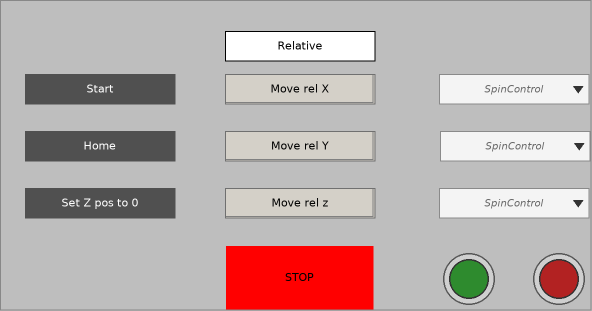
VISUALIZATION goPositionRel  // 592x311
    Button (225,74 150x30), "Move rel X"
        tap POSITION.DoRel_X
    Button (225,131 150x30), "Move rel Y"
        tap POSITION.DoRel_Y
    Button (225,188 150x30), "Move rel z"
        tap POSITION.DoRel_Z
    Rectangle (226,246 147x63), "STOP", colour toggle: GVL.StopALL
        toggle GVL.StopALL
    Rectangle (25,131 150x30), "Home"
        tap INIT.bHome
    Rectangle (25,74 150x30), "Start", colour toggle: INIT.bENCouple
        toggle INIT.bENCouple
    Rectangle (25,188 150x30), "Set Z pos to 0"
        tap POSITION.SetZpos
    SpinControl (439,74 150x30), variable: POSITION.Rel_X
        OnMouseDown: write POSITION.Rel_X via Edit, min 0, max 300
    SpinControl (440,131 150x30), variable: POSITION.Rel_Y
        OnMouseDown: write POSITION.Rel_Y via Edit, min 0, max 300
    SpinControl (439,188 150x30), variable: POSITION.Rel_Z
        OnMouseDown: write POSITION.Rel_Z via Edit, min -80, max 80
    Lamp1 (439,249 60x60), variable: POSITION.Done, style: Lamp-Lamp1-Green
    Lamp1 (529,249 60x60), variable: POSITION.Busy, style: Lamp-Lamp1-Red
    Rectangle (225,31 150x30), "Relative"
END_VISUALIZATION

(* stored: Version 1.1.0.1, ProductVersion 3.1.4022.17
   Visu goPositionRel: Id {edfb47fe-a47b-498c-9a36-c503b3ad69c4} *)
